// TwinCAT 3 PLC project Untitled1
// ProgramVersion: 3.1.4023.0
// libraries:
//   Tc2_MC2, * (Beckhoff Automation GmbH)
//   Tc2_Standard, * (Beckhoff Automation GmbH)
//   Tc2_System, * (Beckhoff Automation GmbH)
//   Tc3_Mc3Definitions, * (Beckhoff Automation GmbH)
//   Tc3_McCoordinatedMotion, * (Beckhoff Automation GmbH)
//   Tc3_Module, * (Beckhoff Automation GmbH)
// project tree:
//   DUTs/ DUT_Test.TcDUT, DUT_Test_1.TcDUT, KinematicsD4.TcDUT
//   GVLs/ GVL_Kinematics.TcGVL
//   / PlcTask.TcTTO
//   POUs/ FB01.TcPOU, MAIN.TcPOU, MotionGroup.TcPOU
// real-time tasks:
//   TASK PlcTask: cycle T#10ms, priority 20, ADS port 350
//   TASK Job Task: cycle default, priority 32
// motion (NC):
//   TASK NC-Task 1 SAF: cycle T#2ms, priority 4, ADS port 501
//   TASK NC-Task 1 SVB: cycle T#10ms, priority 8, ADS port 511
//   AXIS Axis 1 (id 1)
//     General: UnitName=°
//     OtherSettings: AllowMotionCmdToSlave=true
//     encoder EncType=1
//     drive DrvType=5
//       Analog: TorqueSetpointScale=10, ScaleFactorActTorque=0.1
//       TimeComp: TaskDelayCycles=1
//     controller CtrType=1
//       CtrPara: PriorControlFactor=1
//         Observer: BandWidth=20
//   AXIS Axis 2 (id 2)
//     General: UnitName=°
//     OtherSettings: AllowMotionCmdToSlave=true
//     encoder EncType=1
//     drive DrvType=5
//       Analog: TorqueSetpointScale=10, ScaleFactorActTorque=0.1
//       TimeComp: TaskDelayCycles=1
//     controller CtrType=1
//       CtrPara: PriorControlFactor=1
//         Observer: BandWidth=20
//   AXIS Axis 3 (id 3)
//     General: UnitName=°
//     OtherSettings: AllowMotionCmdToSlave=true
//     encoder EncType=1
//     drive DrvType=5
//       Analog: TorqueSetpointScale=10, ScaleFactorActTorque=0.1
//       TimeComp: TaskDelayCycles=1
//     controller CtrType=1
//       CtrPara: PriorControlFactor=1
//         Observer: BandWidth=20
//   AXIS Axis 4 (id 8)
//     OtherSettings: AllowMotionCmdToSlave=true
//     encoder EncType=1
//     drive DrvType=5
//       Analog: TorqueSetpointScale=10, ScaleFactorActTorque=0.1
//     controller CtrType=1
//       CtrPara: PriorControlFactor=1
//         Observer: BandWidth=20
//   AXIS X (id 4)
//     OtherSettings: AllowMotionCmdToSlave=true
//     encoder EncType=1
//     drive DrvType=5
//       Analog: TorqueSetpointScale=10, ScaleFactorActTorque=0.1
//       TimeComp: TaskDelayCycles=1
//     controller CtrType=1
//       CtrPara: PriorControlFactor=1
//         Observer: BandWidth=20
//   AXIS Y (id 5)
//     OtherSettings: AllowMotionCmdToSlave=true
//     encoder EncType=1
//     drive DrvType=5
//       Analog: TorqueSetpointScale=10, ScaleFactorActTorque=0.1
//       TimeComp: TaskDelayCycles=1
//     controller CtrType=1
//       CtrPara: PriorControlFactor=1
//         Observer: BandWidth=20
//   AXIS Z (id 6)
//     OtherSettings: AllowMotionCmdToSlave=true
//     encoder EncType=1
//     drive DrvType=5
//       Analog: TorqueSetpointScale=10, ScaleFactorActTorque=0.1
//       TimeComp: TaskDelayCycles=1
//     controller CtrType=1
//       CtrPara: PriorControlFactor=1
//         Observer: BandWidth=20
//   AXIS C (id 7)
//     OtherSettings: AllowMotionCmdToSlave=true
//     encoder EncType=1
//     drive DrvType=5
//       Analog: TorqueSetpointScale=10, ScaleFactorActTorque=0.1
//       TimeComp: TaskDelayCycles=1
//     controller CtrType=1
//       CtrPara: PriorControlFactor=1
//         Observer: BandWidth=20
// variable links:
//   Untitled1/Untitled1 Instance <-> NC-Task 1 SAF/Axes/Axis 1
//     PlcTask Inputs/GVL_Kinematics.gbKin.ACSRef[1].NcToPlc <-> Outputs/ToPlc
//     PlcTask Outputs/GVL_Kinematics.gbKin.ACSRef[1].PlcToNc <-> Inputs/FromPlc
//   Untitled1/Untitled1 Instance <-> NC-Task 1 SAF/Axes/Axis 2
//     PlcTask Inputs/GVL_Kinematics.gbKin.ACSRef[2].NcToPlc <-> Outputs/ToPlc
//     PlcTask Outputs/GVL_Kinematics.gbKin.ACSRef[2].PlcToNc <-> Inputs/FromPlc
//   Untitled1/Untitled1 Instance <-> NC-Task 1 SAF/Axes/Axis 3
//     PlcTask Inputs/GVL_Kinematics.gbKin.ACSRef[3].NcToPlc <-> Outputs/ToPlc
//     PlcTask Outputs/GVL_Kinematics.gbKin.ACSRef[3].PlcToNc <-> Inputs/FromPlc
//   Untitled1/Untitled1 Instance <-> NC-Task 1 SAF/Axes/Axis 4
//     PlcTask Inputs/GVL_Kinematics.gbKin.ACSRef[4].NcToPlc <-> Outputs/ToPlc
//     PlcTask Outputs/GVL_Kinematics.gbKin.ACSRef[4].PlcToNc <-> Inputs/FromPlc
//   Untitled1/Untitled1 Instance <-> NC-Task 1 SAF/Axes/C
//     PlcTask Inputs/GVL_Kinematics.gbKin.MCSRef[4].NcToPlc <-> Outputs/ToPlc
//     PlcTask Outputs/GVL_Kinematics.gbKin.MCSRef[4].PlcToNc <-> Inputs/FromPlc
//   Untitled1/Untitled1 Instance <-> NC-Task 1 SAF/Axes/X
//     PlcTask Inputs/GVL_Kinematics.gbKin.MCSRef[1].NcToPlc <-> Outputs/ToPlc
//     PlcTask Outputs/GVL_Kinematics.gbKin.MCSRef[1].PlcToNc <-> Inputs/FromPlc
//   Untitled1/Untitled1 Instance <-> NC-Task 1 SAF/Axes/Y
//     PlcTask Inputs/GVL_Kinematics.gbKin.MCSRef[2].NcToPlc <-> Outputs/ToPlc
//     PlcTask Outputs/GVL_Kinematics.gbKin.MCSRef[2].PlcToNc <-> Inputs/FromPlc
//   Untitled1/Untitled1 Instance <-> NC-Task 1 SAF/Axes/Z
//     PlcTask Inputs/GVL_Kinematics.gbKin.MCSRef[3].NcToPlc <-> Outputs/ToPlc
//     PlcTask Outputs/GVL_Kinematics.gbKin.MCSRef[3].PlcToNc <-> Inputs/FromPlc
//   Untitled1/Untitled1 Instance <-> NC-Task 1 SAF/Objects/Group1 (MC Group Coordinated Motion)
//     PlcTask Inputs/GVL_Kinematics.gbKin.GroupRef.NcToPlc <-> Group Outputs/ToPLC
//     PlcTask Outputs/GVL_Kinematics.gbKin.GroupRef.PlcToNc <-> Group Inputs/FromPLC

CONFIGURATION Untitled1
    RESOURCE PLC ON TwinCAT3
        TASK PlcTask(INTERVAL := T#10ms, PRIORITY := 20);
        PROGRAM MAIN WITH PlcTask : MAIN;
    END_RESOURCE
END_CONFIGURATION

// ---- DUTs/DUT_Test.TcDUT
TYPE DUT_Test :
STRUCT
	value: BOOL;
	abc: DUT_Test_1;
END_STRUCT
END_TYPE

// ---- DUTs/DUT_Test_1.TcDUT
TYPE DUT_Test_1 :
STRUCT
	a : BOOL;
	b : REAL;
	c : string(200);
END_STRUCT
END_TYPE

// ---- DUTs/KinematicsD4.TcDUT
TYPE KinematicsD4 :
STRUCT
	GroupRef: AXES_GROUP_REF;
	ACSRef: ARRAY[1..4] OF Axis_Ref;
	MCSRef: ARRAY[1..4] OF Axis_Ref;
END_STRUCT
END_TYPE

// ---- GVLs/GVL_Kinematics.TcGVL
VAR_GLOBAL
	gbKin : KinematicsD4;
END_VAR

// ---- POUs/MAIN.TcPOU
PROGRAM MAIN
VAR
	bTest_bool  AT %I* :  BOOL;
	iTest_int: INT;
	sTest_string: STRING;	
	DutTest: Dut_Test;
	fb_test: FB01;
END_VAR


sTest_String:='beckhoff';

bTest_bool:=TRUE;
DutTest.abc.a:=TRUE;
fb_test(input1:= , output1=> );

MotionGroup();

END_PROGRAM

// ---- POUs/FB01.TcPOU
FUNCTION_BLOCK FB01
VAR_INPUT
	input1: BOOL;
END_VAR
VAR_OUTPUT
	output1: bool;
END_VAR
VAR
END_VAR

output1:=input1;

END_FUNCTION_BLOCK

// ---- POUs/MotionGroup.TcPOU
PROGRAM MotionGroup
VAR
	_fb_AddAxisTOGroup: ARRAY[1..iAxesCount] OF MC_AddAxisToGroup;
	i: INT;
	
	_fb_GroupEnable: MC_GroupEnable;
	_fb_GroupDisable: MC_GroupDisable;
	_fb_GroupReadError: MC_GroupReadError;
	_fb_GroupReadStatus: MC_GroupReadStatus;
	_fb_GroupReset: MC_GroupReset;
	_fb_GroupSetOverride: MC_GroupSetOverride;
	_fb_RemoveAxisFromGroup: MC_RemoveAxisFromGroup;
	_fb_SetCoordinateTransform: MC_SetCoordinateTransform;
	_fb_TrackConveyorBelt: MC_TrackConveyorBelt;
	_fb_UngroupAllAxes: MC_UngroupAllAxes;
	_fb_MoveLinearAbsolutePreparation: MC_MoveLinearAbsolutePreparation;
	
	_Buffer: ARRAY[1..4096] OF BYTE ;
	_PathData: MC_PATH_DATA_REF(ADR(_Buffer),SIZEOF(_buffer));
	
	_arPosition: ARRAY[1..4] OF MC_LREAL :=[100,100,0,90];
	_PositionCount: UDINT :=4;
	_Velocity: MC_LREAL:=10;
	_Accel: MC_LREAL:=100;
	_Decel: MC_LREAL:=100;
	_Jerk: MC_LREAL:=1000;
	_BufferMode: MC_BUFFER_MODE := mcBlendinglow;
	_TransitionMode: MC_TRANSITION_MODE:= mcTransModeCornerDistanceAdvanced;
	_arTransitionPara: ARRAY[1..2] OF MC_LReal :=[10,10];
	_TransitionParaCount: UDINT:=2;
	_InvokeId: UDINT;
	_PathDataFilledRows: UDINT;
	_PathDataOccupiedBuffer: UDINT;
	
	
	_bWritePosition: BOOL;
	_rt_WritePosition: R_trig;
	
	_fb_MovePath: MC_MovePath;
	
END_VAR
VAR CONSTANT
	iAxesCount: INT:=4;
END_VAR

_fb_AddAxisTOGroup[1].IdentInGroup := MCS_X;
_fb_AddAxisTOGroup[2].IdentInGroup := MCS_Y;
_fb_AddAxisTOGroup[3].IdentInGroup := MCS_Z;
_fb_AddAxisTOGroup[4].IdentInGroup := MCS_C1;
FOR i:=1 TO iAxesCount DO
_FB_AddAxisTOGroup[i](
	AxesGroup:= gbkin.groupRef, 
	Axis:= gbkin.MCSRef[i], 
	Execute:= , );
END_FOR;

_fb_GroupEnable(
	AxesGroup:= gbkin.groupRef, 
	Execute:=,  );
	
_fb_GroupReadError(
	AxesGroup:= gbkin.groupRef, 
	Enable:= TRUE, );

_fb_GroupReadStatus(
	AxesGroup:= gbkin.groupRef, 
	Enable:= TRUE, );
	

_fb_GroupReset(
	AxesGroup:= gbkin.groupRef, 
	Execute:= ,  );	

_PathData(FilledRows=> _PathDataFilledRows, OccupiedBuffer=> _PathDataOccupiedBuffer);	
_rt_WritePosition(CLK:= _bWritePosition, Q=> );


IF _rt_WritePosition.Q THEN
	_fb_MoveLinearAbsolutePreparation(
		PathData:= _PathData, 
		Position:= ADR(_arPosition), 
		PositionCount:= _PositionCount, 
		Velocity:= _Velocity, 
		Acceleration:= _Accel, 
		Deceleration:= _Decel, 
		Jerk:= _Jerk, 
		BufferMode:= _BufferMode, 
		TransitionMode:= _TransitionMode, 
		TransitionParameter:= ADR(_arTransitionPara), 
		TransitionParameterCount:= _TransitionParaCount, 
		InvokeId:= _InvokeId, 
		Error=> , 
		ErrorId=> );
END_IF	
	
_fb_MovePath(
	AxesGroup:= gbkin.groupRef, 
	PathData:= _PathData, 
	Execute:= , 
 );

END_PROGRAM
